// TIA Portal V19 export
FUNCTION "Komm_PNOZ" : Void   // FC360, STL
TITLE = Kommunikation Pilz-PNOZ <--> PLC
{ S7_Optimized_Access := 'FALSE' }
// stored: AutoNumber false
   VAR_TEMP
      Checksum : Word;
      ReturnValue : Int;
      count : Byte;
   END_VAR
BEGIN

NETWORK
TITLE = Aktivierung der Kommunikation

      AN    "DB_PNOZ_Comm".connection.activate;
      A     "E_T_ErrQ";
      S     "DB_PNOZ_Comm".connection.activate;


NETWORK
TITLE = OUTPUT --> PNOZ
// siehe Handbuch
// "PNOZmulti_2_Com_Interf_Man_1002971-de-03.pdf"
// Set Header   (Kap. 5.5)
      L     16#05;
      T     "DB_PNOZ_IN_Out".Out.Header[0];

      L     16#15;
      T     "DB_PNOZ_IN_Out".Out.Header[1];

      L     16#00;
      T     "DB_PNOZ_IN_Out".Out.Header[2];

      L     16#26;  // Anzahl Nutzdaten +5  = 38 dez
      T     "DB_PNOZ_IN_Out".Out.Header[3];

      L     16#5C;  // Anforderungs-Nr
      T     "DB_PNOZ_IN_Out".Out.Header[4];

      L     16#00;
      T     "DB_PNOZ_IN_Out".Out.Header[5];  // Control Byte Bit 0..2 Watchdog

      L     16#00;
      T     "DB_PNOZ_IN_Out".Out.Header[6];

      L     16#00;  // immer 0x00
      T     "DB_PNOZ_IN_Out".Out.Header[7];

      L     16#10;
      T     "DB_PNOZ_IN_Out".Out.Endekennung;

// Set Vitual OUTput - je nach Projekt
      A     "E_T_Q_Not-Halt";
// alle Schütze müssen abgefallen sein
      A     "E_RM_NH_Dkl";
      A     "E_RM_NH_FP_CM01.GP01";
      A     "E_RM_NH_FP_CM01.GP04";
      A     "E_RM_NH_Pumpen";
      =     "DB_PNOZ_IN_Out".Out.T_NH_Quitt;
// Freigabe Automatik
      A     "E_Frg_Auto";
      =     "DB_PNOZ_IN_Out".Out.Frg_Automatik;

      CLR;
      =     "DB_PNOZ_IN_Out".Out.VirtualOutput[16];
// ...
      =     "DB_PNOZ_IN_Out".Out.VirtualOutput[127];

// Berechnung der Checksumme (4+ .. 39)

      LAR1  P#48.0;  // fix 44 (IN) + 4

      L     "DB_PNOZ_IN_Out".Out.Header[4];  //Start
      T     #Checksum;

      L     35;  // fix: 39 - 4
T_CS: T     #count;
      OPN   "DB_PNOZ_IN_Out";
      +AR1  P#1.0;
      L     #Checksum;
      L     DBB [AR1, P#0.0];
      +I;
      T     #Checksum;

      L     #count;  //Schleifenzähler
      LOOP  T_CS;

      L     16#00;
      L     #Checksum;
      AW    16#00FF;
      -I;
      T     "DB_PNOZ_IN_Out".Out.Checksum;



NETWORK
TITLE = Umkopieren
// Sende-/Empfangsdaten umkopieren

      A     "DB_PNOZ_Comm".RECEIVE.NDR;
      R     "DB_PNOZ_Comm".RECEIVE.NDR;
      JCN   Send;

      CALL  BLKMOV
      ( SRCBLK  := "DB_PNOZ_Receive".In,
        RET_VAL := #ReturnValue,
        DSTBLK  := "DB_PNOZ_IN_Out".In
      );

Send: A     "DB_PNOZ_Comm".SEND.Busy;
      JC    no_Send_DATA;

      CALL  BLKMOV
      ( SRCBLK  := "DB_PNOZ_IN_Out".Out,
        RET_VAL := #ReturnValue,
        DSTBLK  := "DB_PNOZ_Send".Out
      );

no_Send_DATA:NOP   0;

NETWORK
TITLE = Sprungverteiler

      L     "DB_PNOZ_Comm".Global_Status;
      JL    LSTX;
      JU    OFF;  // 0: Aus
      JU    CONN;  // 1: Verbindungsaufbau
      JU    WRIT;  // 2: Schreiben
      JU    READ;  // 3: Lesen
      JU    DISC;  // 4:Verbindungsabbau
      JU    ERR;  // 5: Fehler
LSTX: JU    ende;

//*
// wait for user input (activate / deactivate communication)
// - if activate change for 0 to 1
//    => status is set to 1 (connect) and all status-values are set to default
// - if activate change for 1 to 0
//    => status is set to 4 (disconnect)
//-

OFF:  A     "DB_PNOZ_Comm".connection.activate;
      AN    "DB_PNOZ_Comm".connection.established;
      JCN   OFF1;

// Aktivieren
      SET;
      S     "DB_PNOZ_Comm".connection.established;

      L     1;  // Verbindungsaufbau
      T     "DB_PNOZ_Comm".Global_Status;

// init
      SET;
      R     "DB_PNOZ_Comm".CONNECT.Request;
      R     "DB_PNOZ_Comm".CONNECT.Done;
      R     "DB_PNOZ_Comm".CONNECT.Error;

      R     "DB_PNOZ_Comm".SEND.Request;
      R     "DB_PNOZ_Comm".SEND.Done;
      R     "DB_PNOZ_Comm".SEND.Error;

      S     "DB_PNOZ_Comm".RECEIVE.EN_R;  // immer 1
      R     "DB_PNOZ_Comm".RECEIVE.NDR;
      R     "DB_PNOZ_Comm".RECEIVE.Error;

      R     "DB_PNOZ_Comm".DISCONNECT.Request;
      R     "DB_PNOZ_Comm".DISCONNECT.Done;
      R     "DB_PNOZ_Comm".DISCONNECT.Error;

      JU    ende;

// Deaktivieren
OFF1: AN    "DB_PNOZ_Comm".connection.activate;
      A     "DB_PNOZ_Comm".connection.established;
      JCN   ende;

      SET;
      R     "DB_PNOZ_Comm".connection.established;
      R     "DB_PNOZ_Comm".CONNECT.Done;
      R     "DB_PNOZ_Comm".SEND.Done;
      R     "DB_PNOZ_Comm".RECEIVE.NDR;

      L     4;  // Verbindungsabbau
      T     "DB_PNOZ_Comm".Global_Status;

      JU    ende;


NETWORK
TITLE = Verbindungsaufbau
// call FB65 (TCON) as long as status = 1 (connect)
//  - if connection_1 is established (TCON_DONE=1) change to status=2 (send)
//  - if an error occurs (TCON_ERR=1) change to status=5 (error)
CONN: L     2;
      T     "DB_PNOZ_Comm".CONNECT.ID;
      T     "DB_PNOZ_Comm".Connection_Param.local_device_id;

      CALL  TCON, "TCON_DI"
      ( REQ     := "DB_PNOZ_Comm".CONNECT.Request,
        ID      := "DB_PNOZ_Comm".CONNECT.ID,
        DONE    := "DB_PNOZ_Comm".CONNECT.Done,
        BUSY    := "DB_PNOZ_Comm".CONNECT.Busy,
        ERROR   := "DB_PNOZ_Comm".CONNECT.Error,
        STATUS  := "DB_PNOZ_Comm".CONNECT.Status,
        CONNECT := "PNOZ_Connection_DB"
      );

      SET;
      S     "DB_PNOZ_Comm".CONNECT.Request;

      A     "DB_PNOZ_Comm".CONNECT.Done;
      R     "DB_PNOZ_Comm".CONNECT.Done;
      R     "DB_PNOZ_Comm".SEND.Request;
      JC    to_S;

      L     "DB_PNOZ_Comm".CONNECT.Status;
      L     16#80A3;  //Verbindung gibt's schon
      ==I;
      A     "DB_PNOZ_Comm".CONNECT.Error;
      R     "DB_PNOZ_Comm".DISCONNECT.Request;
      JC    to_D;

      A     "DB_PNOZ_Comm".CONNECT.Error;
      JC    to_E;

      JU    ende;

to_S: L     2;  // --> Senden
      T     "DB_PNOZ_Comm".Global_Status;
      JU    ende;

to_D: L     4;  // --> Verbindungsabbau
      T     "DB_PNOZ_Comm".Global_Status;
      JU    ende;


to_E: L     5;  // --> Fehler
      T     "DB_PNOZ_Comm".Global_Status;

      JU    ende;


NETWORK
TITLE = Schreiben --> PNOZ
// call FB63 (TSEND) as long as status = 2 (send)
//  - if send is complete (TSEND_DONE=1) change to status=3 (receive)
//  - if an error occurs (TSEND_ERR=1)
//    - if TSEND_STATUS='80A1' or '80C4' stay at status=2 and try to send again
//    - if TSEND_STATUS<>'80A1' or '80C4' change to status=5 (error)
WRIT: L     43;  //fix PNOZ
      T     "DB_PNOZ_Comm".SEND.Length;

      L     "DB_PNOZ_Comm".CONNECT.ID;
      T     "DB_PNOZ_Comm".SEND.ID;

      CALL  TSEND, "TSEND_DI"
      ( REQ    := "DB_PNOZ_Comm".SEND.Request,
        ID     := "DB_PNOZ_Comm".SEND.ID,
        LEN    := "DB_PNOZ_Comm".SEND.Length,
        DONE   := "DB_PNOZ_Comm".SEND.Done,
        BUSY   := "DB_PNOZ_Comm".SEND.Busy,
        ERROR  := "DB_PNOZ_Comm".SEND.Error,
        STATUS := "DB_PNOZ_Comm".SEND.Status,
        DATA   := "DB_PNOZ_Send".Out
      );

      SET;
      S     "DB_PNOZ_Comm".SEND.Request;

      A     "DB_PNOZ_Comm".SEND.Done;
      R     "DB_PNOZ_Comm".SEND.Done;
      S     "DB_PNOZ_Comm".RECEIVE.EN_R;
      JC    toRV;

      L     16#80A1;  //Kommunikationsfehler
      L     "DB_PNOZ_Comm".SEND.Status;
      ==I;
      O(;
      L     16#80C4;  //Temporärer Kommunikationsfehler
      ==I;
      );
      A     "DB_PNOZ_Comm".SEND.Error;
      R     "DB_PNOZ_Comm".SEND.Request;  // --> nochmal versuchen
      JC    ende;

      A     "DB_PNOZ_Comm".SEND.Error;
      JC    SDER;

      JU    ende;

toRV: L     3;
      T     "DB_PNOZ_Comm".Global_Status;
      JU    ende;

SDER: L     5;
      T     "DB_PNOZ_Comm".Global_Status;
      JU    ende;


NETWORK
TITLE = Lesen <-- PNOZ
// call FB64 (TRCV) as long as status = 3 (receive)
//  - if new data is received (TSEND_NDR=1) change to status=2 (receive)
//    and increment send_values
//  - if an error occurs (TRCV_ERR=1)
//    - if TRCV_STATUS='80A1' or '80C4' change to status=2 and try to send
//    - if TRCV_STATUS<>'80A1' or '80C4' change to status=5 (error)
READ: L     43;  //fix PNOZ
      T     "DB_PNOZ_Comm".RECEIVE.Length;

      L     "DB_PNOZ_Comm".CONNECT.ID;
      T     "DB_PNOZ_Comm".RECEIVE.ID;

      CALL  TRCV, "TRCV_DI"
      ( EN_R     := "DB_PNOZ_Comm".RECEIVE.EN_R,
        ID       := "DB_PNOZ_Comm".RECEIVE.ID,
        LEN      := "DB_PNOZ_Comm".RECEIVE.Length,
        ADHOC    := "DB_PNOZ_Comm".RECEIVE.ADHOC,
        NDR      := "DB_PNOZ_Comm".RECEIVE.NDR,
        BUSY     := "DB_PNOZ_Comm".RECEIVE.Busy,
        ERROR    := "DB_PNOZ_Comm".RECEIVE.Error,
        STATUS   := "DB_PNOZ_Comm".RECEIVE.Status,
        RCVD_LEN := "DB_PNOZ_Comm".RECEIVE.Receive_Length,
        DATA     := "DB_PNOZ_Receive".In
      );

      A     "DB_PNOZ_Comm".RECEIVE.NDR;
      JC    toSD;

      L     16#80A1;  //Kommunikationsfehler
      L     "DB_PNOZ_Comm".RECEIVE.Status;
      ==I;
      O(;
      L     16#80C4;  //Temporärer Kommunikationsfehler
      ==I;
      );
      A     "DB_PNOZ_Comm".RECEIVE.Error;
      R     "DB_PNOZ_Comm".RECEIVE.Error;
      JC    toSD;

      A     "DB_PNOZ_Comm".RECEIVE.Error;
      JC    RVER;

      JU    ende;

toSD: L     2;
      T     "DB_PNOZ_Comm".Global_Status;
      SET;
      R     "DB_PNOZ_Comm".SEND.Request;
      JU    ende;

RVER: L     5;
      T     "DB_PNOZ_Comm".Global_Status;
      JU    ende;


NETWORK
TITLE = Verbindungsabbau
// call FB66 (TDISCON) as long as status = 4 (disconnect)
//  - if connection_1 is disconnected (TDISCON_DONE=1) change to status=0 (init)
//  - if an error occurs (TDISCON_ERR=1) change to status=5 (error)
DISC: L     "DB_PNOZ_Comm".CONNECT.ID;
      T     "DB_PNOZ_Comm".DISCONNECT.ID;

      CALL  TDISCON, "TDISCON_DI"
      ( REQ    := "DB_PNOZ_Comm".DISCONNECT.Request,
        ID     := "DB_PNOZ_Comm".DISCONNECT.ID,
        DONE   := "DB_PNOZ_Comm".DISCONNECT.Done,
        BUSY   := "DB_PNOZ_Comm".DISCONNECT.Busy,
        ERROR  := "DB_PNOZ_Comm".DISCONNECT.Error,
        STATUS := "DB_PNOZ_Comm".DISCONNECT.Status
      );

      SET;
      S     "DB_PNOZ_Comm".DISCONNECT.Request;

      A     "DB_PNOZ_Comm".DISCONNECT.Done;
      R     "DB_PNOZ_Comm".DISCONNECT.Done;
      R     "DB_PNOZ_Comm".connection.activate;
      R     "DB_PNOZ_Comm".connection.established;
      JC    to_O;

      A     "DB_PNOZ_Comm".DISCONNECT.Error;
      JC    toE;

      JU    ende;

to_O: L     0;  // --> OFF
      T     "DB_PNOZ_Comm".Global_Status;
      JU    ende;

toE:  L     5;  // --> Fehler
      T     "DB_PNOZ_Comm".Global_Status;
      JU    ende;


NETWORK
TITLE = Fehler
ERR:  SET;
      R     "DB_PNOZ_Comm".connection.activate;
      R     "DB_PNOZ_Comm".connection.established;

      L     0;  // --> OFF
      T     "DB_PNOZ_Comm".Global_Status;

ende: BE;

END_FUNCTION
